(*
Nazwa:			GVL_Recipe
Opis:			Zmienne recepturowe tylko do wizualizacji
Wersja:			v0.2
Data:			2024-02-20
Autor:			MK
Urzadzenia:		
Konfiguracja:	
Info:
Zmiany:
- 20240220 [DP] Poprawki przed nowa wizką
*)
VAR_GLOBAL
	(*Legenda dla wizki :
		[H] - Hidden, prawdopodobnie nie potrzebne
		[I] - Info, informacja,
		[L] - Later, do zrobienia później, być może do przerobienia
		Uprawienia:
		brak opisu - operator
		[m] - Meechanik i powyżej
		[t] - Technolog i powyżej
		[s] - Serwis i powyżek
		[a] - Admin			
	*)	
	
	//Sorter nasadek, typ produktu	
	iCapSorterProductType										: INT		:= 2; 		//		Typ produktu: 0- kule/fliptopy, 1- pompki, 2- disctop, 3-airless, 4-decoration cap (wyłączone podcisnienie na załapywarce), 5- decoration cap with new gripper (wyłączone podcisnienie + nowy program do robota)
	uiCapSorterIndexShow										: UDINT		:= 5;		//		Index produktu	
	bPresenceBottleEnableShow									: BOOL;					//		Sprawdzanie butelki w formatce

//--------------------------------------CapSorterTransporter-----------------------------------------------------------------------------------------------------------------------------	
	// Sorter nasadek, transporter zasobnika
	bCapSorterTransporterEnableShow								: BOOL;					//		Aktywacja
	iCapSorterTransporterTankConveyorVelocityShow				: INT		:= 1200;	//		Prędkość 							| [%] (1.0-100.0)
	iCapSorterTransporterStartDelayTimeShow						: INT		:= 100;		//		Timer do załączania 				| [ms] (0.0-10_000.0)
	udiCapSorterTransporterTimeProductOnSensorBeforeBrushShow	: UDINT		:= 150;		//		Timer pracy							| [ms] (0.0-10_000.0)
	iCapSorterTransporterEmptyingConveyorSpeedShow				: INT		:= 25;		// 		Prędkość, opróżnianie 				| [%] (1.0-100.0)
	iCapSorterTransporterVolumeOfCapsShow						: INT		:= 330;		//		Odłegłość do zamknięć, ostrzeżenie 	| [mm] (0.0-10_000.0)

//---------------------------------------CapSorterWheel----------------------------------------------------------------------------------------------------------------------------	
	// Sorter nasadek, stól
	bCapSorterWheelEnableShow									: BOOL;					//		Aktywacja
	lrCapSorterWheelMoveAccelerationEmptyTableShow				: LREAL		:= 5000;	//		Dynamika rozpędzania - pusty 		| [obr/min²], (1.0-100_000.0) 
	lrCapSorterWheelMoveDecelerationEmptyTableShow				: LREAL		:= 5000;    //		Dynamika spowalniania - pusty 		| [obr/min²] (1.0-100_000.0) 
	lrCapSorterWheelMoveSpeedEmptyTableShow						: LREAL		:= 334;     //		Prędkość - pusty 					| [obr/min] (1.0-10_000.0)                
	lrCapSorterWheelMoveAngleEmptyTableShow						: LREAL		:= 20;      //		Kąt - pusty 						| [obr/min] (0.0-360.0)                        
	lrCapSorterWheelJerkAngleEmptyTableShow						: LREAL		:= 15000;   //		Zryw - pusty 						| [obr/min³] (1.0-1_000_000)                  
	iCapSorterWheelWaitingAfterRotationEmptyTableShow			: INT		:= 100;     //		Czas stabilizacji - pusty 			| [ms] (0.0-1_000)                 
	
	lrCapSorterWheelMoveAccelerationFullTableShow				: LREAL		:= 5000;	//		Dynamika rozpędzania - pełny 		| [obr/min²], (1.0-100_000.0) 
	lrCapSorterWheelMoveDecelerationFullTableShow				: LREAL		:= 5000;    //		Dynamika spowalniania - pełny 		| [obr/min²] (1.0-100_000.0) 
	lrCapSorterWheelMoveSpeedFullTableShow						: LREAL		:= 334;     //		Prędkość - pełny 					| [obr/min] (1.0-10_000.0)                
	lrCapSorterWheelMoveAngleFullyTableShow						: LREAL		:= 6;       //		Kąt - pełny 						| [obr/min] (0.0-360.0)                        
	lrCapSorterWheelJerkAngleFullTableShow						: LREAL		:= 15000;   //		Zryw - pełny 						| [obr/min³] (1.0-1_000_000)                  
	iCapSorterWheelWaitingAfterRotationFullTableShow			: INT		:= 30;      //		Czas stabilizacji - pełny 			| [ms] (0.0-1_000)                 
	
	lrCapSorterWheelMoveAccelerationHalfFullTableShow			: LREAL		:= 5000;	//		Dynamika rozpędzania - półpełny 	| [obr/min²], (1.0-100_000.0) 
	lrCapSorterWheelMoveDecelerationHalfFullTableShow			: LREAL		:= 5000;    //		Dynamika spowalniania - półpełny 	| [obr/min²] (1.0-100_000.0) 
	lrCapSorterWheelMoveSpeedHalfFullTableShow					: LREAL		:= 334;     //		Prędkość - półpełny 				| [obr/min] (1.0-10_000.0)                
	lrCapSorterWheelMoveAngleHalfFullyTableShow					: LREAL		:= 12;      //		Kąt - półpełny						| [obr/min] (0.0-360.0)                        
	lrCapSorterWheelJerkAngleHalfFullTableShow					: LREAL		:= 15000;   //		Zryw - półpełny 					| [obr/min³] (1.0-1_000_000)                  
	iCapSorterWheelWaitingAfterRotationHalfFullTableShow		: INT		:= 50;      //		Czas stabilizacji - półpełny 		| [ms] (0.0-1_000)               
	
//-------------------------------------CapSorterCamera------------------------------------------------------------------------------------------------------------------------------	                                                    	
	// Sorter nasadek, system wizyjny
	
    bCapSorterCameraEnableShow									: BOOL; 				//	[H]	Aktywacja                            	
	
//-----------------------------------------CapSorterRobot--------------------------------------------------------------------------------------------------------------------------	
	// Sorter nasadek, robot
	bCapSorterRobotEnableShow									: BOOL;					//		Aktywacja
                                                                                                                           	
	lrCapSorterRobotPlace1PositionXShow							: LREAL;				//		Offset odkładania 1, X 			| [mm]	((-100.0)-100.0)       
	lrCapSorterRobotPlace1PositionYShow							: lreal;    			//		Offset odkładania 1, Y 			| [mm]	((-100.0)-100.0)       
	lrCapSorterRobotPlace1PositionZShow							: lreal;    			//		Offset odkładania 1, Z 			| [mm]	((-100.0)-100.0)       
	lrCapSorterRobotPlace1PositionCShow							: lreal;    			//		Offset odkładania 1, C 			| [° ]	((-360.0)-360.0)                 
	iCapSorterRobotPickElevationShow							: INT;					//		Punkt nad poz. Pick				| [mm]	(30-1000)
	iCapSorterRobotPickTimeShow									: INT;					//		Czas przyssania					| [ms]	(0-10_000)
	iCapSorterRobotVacuumActivationShow							: INT;					//		Czas przed przyssaniem			| [ms]	(0-1000)
	iCapSorterRobotVacuumOffShow								: INT;					//		Czas przed oddmuchem			| [ms]	(0-1000)
	iCapSorterRobotPlaceTimeShow								: INT;					//		Czas oddmuchu					| [ms]	(0-1000)
	iCapSorterRobotTCP_PlaceOffsetShow							: INT;					//		Wysokość od TCP do p. odłożenia	| [mm]	(0-1000)									
	iCapSorterRobotAccelerationDecelerationShow					: INT;					//		Dynamika rozpędzania/hamowania	| [%]	(20-100)
	iCapSorterRobotGripperWatchdogShow							: INT;					//		Czas sprawdzania silownika		| [ms]	(0-1000)
	iCapSorterRobotParalaxCorrectionShow						: INT;					//		Korekta paralaxy				| [mm]	(0-100)
	
	iCapSorterRobotNumberToolShow								: INT;					//		Numer narzędzia					| 		(0-10)
	iCapSorterRobotPickPositionZShow							: INT;					//		Wysokość pobierania 			| [mm]	(0-200)
	iCapSorterRobotTCP_Lenght									: INT;					//		Długość chwytaka				| [mm]	(10-100)
	iCapSorterRobotProductDiametr								: INT;					//		Średnica nasadki				| [mm] 	(10-100)
	
//----------------------------------------CapSorterIntermediateTransporter---------------------------------------------------------------------------------------------------------------------------
	// Sorter nasadek, transporter zasypowy
	bCapSorterIntermediateTransporterEnableShow					: BOOL;					//		Aktywacja
	iCapSorterIntermediateTransporterAutoSpeedShow				: INT		:= 20;		//		Prędkość 					| [%] (1.0-100.0)
	iCapSorterIntermediateTransporterManualSpeedShow			: INT		:= 30;		//		Prędkość, manual 			| [%] (1.0-100.0)
	iCapSorterIntermediateTransporterEmptyingSpeedShow			: INT		:= 50;		//		Prędkość, opróżnianie 		| [%] (1.0-100.0)
	iCapSorterIntermediateTransporterDelayCountTimeShow			: INT		:= 100;		//		Timer pracy					| [ms]	(0.0-100_000.0)
	iCapSorterIntermediateTransporterReverseTimeShow			: INT		:= 4000;	//		Timer odwróconej pracy 		| [ms] (0.0-10_000.0)
	udiCapSorterIntermediateTransporterTimeProductOnSensorShow	: UDINT		:= 1800;	//		Czas produktu na czujniku 	| [ms] (0.0-10_000.0)	
	lrCapSorterIntermediateTransporterWheelAngleShow			: LREAL		:= 6;		//		Kąt zasypu 					| [°] (1.0-360.0)
	lrCapSorterIntermediateTransporterItemsSetValueShow			: LREAL	;				// 		Ilość detali na kołe		| []
	
//----------------------------------------CapSorterIntermediateBrush---------------------------------------------------------------------------------------------------------------------------
	//Sorter nasadek, szczotka transportera
	bCapSorterIntermediateBrushEnableShow						: BOOL;					//		Aktywacja
	iCapSorterIntermediateBrushAutoSpeedShow					: INT		:= 30;		//		Prędkość  					| [%] (0.0-100.0)
	iCapSorterIntermediateBrushManualSpeedShow					: INT		:= 30;		//		Prędkość, manual 			| [%] (0.0-100.0)
	iCapSorterIntermediateBrushEmptyingSpeedShow				: INT		:= 30;		//		Prędkość, opróżnianie 		| [%] (0.0-100.0)
	lrCapSorterIntermediateBrushPositionHeightSVShow			: LREAL		:= 45;		//		Wysokość 					| [mm] (0.0-10_000.0)

//----------------------------------------CapSorterBrush1OnWheel---------------------------------------------------------------------------------------------------------------------------
	// Sorter nasadek, szczotka stolu 1
	bCapSorterBrush1OnWheelEnableShow							: BOOL;					//		Aktywacja
	iCapSorterBrush1OnWheelAutoSpeedShow						: INT		:= 30;		//		Prędkość 					| [%] (0.0-100.0)
	iCapSorterBrush1OnWheelManualSpeedShow						: INT		:= 30;		//		Prędkość, manual 			| [%] (0.0-100.0)
	iCapSorterBrush1OnWheelEmptyingSpeedShow					: INT		:= 30;		//		Prędkość, opróżnianie 		| [%] (0.0-100.0)
	lrCapSorterBrush1OnWheelPositionHeightSVShow				: LREAL		:= 45;		//		Wysokość 					| [mm] (0.0-10_000.0)
	
//----------------------------------------CapSorterBrush2OnWheel----------------------------------------------------------------------------------
	// Sorter nasadek, szczotka stolu 2
	bCapSorterBrush2OnWheelEnableShow							: BOOL;					//		Aktywacja
	iCapSorterBrush2OnWheelAutoSpeedShow						: INT		:= 30;		//		Prędkość 					| [%] (0.0-100.0)
	iCapSorterBrush2OnWheelManualSpeedShow						: INT		:= 30;		//		Prędkość, manual 			| [%] (0.0-100.0)
	iCapSorterBrush2OnWheelEmptyingSpeedShow					: INT		:= 30;		//		Prędkość, opróżnianie 		| [%] (0.0-100.0)
	lrCapSorterBrush2OnWheelPositionHeightSVShow				: LREAL		:= 45;		//		Wysokość 					| [mm] (0.0-10_000.0)

//------------------------------------------CapFeeder-------------------------------------------------------------------------------------------------------------------------	
	// Sorter nasadek, 
	bCapSorterFeederEnableShow									: BOOL;					//		Aktywacjaa
	bCapSorterFeederEnableTubeError								: BOOL;					// 		Aktywacja błedu słomki
	lrCapSorterFeederMover1InputPositionShow					: LREAL;				//		Pozycja wkładania, wózek 1 	| [mm] (?-?)
	lrCapSorterFeederMover2InputPositionShow					: LREAL;				//		Pozycja wkładania, wózek 2 	| [mm] (?-?)
	lrCapSorterFeederMover1OutputPositionShow					: LREAL;				//		Pozycja wyjmowania, wózek 1 | [mm] (?-?)
	lrCapSorterFeederMover2OutputPositionShow					: LREAL;				//		Pozycja wyjmowania, wózek 2 | [mm] (?-?)
	lrCapSorterFeederSlotDistanceShow							: LREAL;				//		Offset wkładania			| [mm] (?-?)			Old-(Odstęp między pozycjami kładzenia)
	lrCapSorterFeederMoverSpeedShow								: LREAL;				//		Prędkość				 	| [%] (0.0-100.0)
	lrCapSorterFeederMoverAccelerationShow						: LREAL;				//		Przyspieszenie 				| [mm/s²] 
	lrCapSorterFeederMoveJerkShow								: LREAL;				//		Zryw						| [mm/s³]

//-------------------------------------------------------------------------------------------------------------------------------------------------------------------	
	//CapPreScrewer		
	bCapSorterPreScrewerEnableShow								: BOOL;					// 		Aktywacja
	bCapSorterPreScrewerPicker1EnableShow						: BOOL;					// 		Aktywacja	
	bCapSorterPreScrewerPicker2EnableShow						: BOOL;					// 		Aktywacja
	bCapSorterPreScrewerPicker3EnableShow						: BOOL;					// 		Aktywacja	
	bCapSorterPreScrewerPicker4EnableShow						: BOOL;					// 		Aktywacja
	//Oś Z
	lrCapSorterPreScrewerPickZPositionShow						: LREAL;				//		Wysokość pobierania						| [mm]	
	lrCapSorterPreScrewerCatcherReleseShow						: LREAL;				//		nie używamy Wysokość otwierania chwytaka nakrętek	| [mm]		
	lrCapSorterPreScrewerCapCatcherZPositionShow				: LREAL;				//		Wysokość zamykania nakrętkek			| [mm]
	lrCapSorterPreScrewerTopZPositionShow						: LREAL;				//		Pozycja górna ośi Z						| [mm] 	
	lrCapSorterPreScrewerCartesianCatchZPositionShow			: LREAL; 				//      Wait Position
	lrCapSorterPreScrewerStrawCatcherZPositionShow				: LREAL;				//		Wysokość otwierania łapaczy słomek		| [mm]	
	LrCapSorterPreScrewerCheckStrawCatcherActuatorZPosition		: LREAL;				//		Wysokość sparawdzania cofania łapaczy słomek	| [mm]	
	lrCapSorterPreScrewerScrewerStartZPositionShow				: LREAL;				//		Wysokość początku zakręcania			| [mm]	
	lrCapSorterPreScrewerGripperOpenPositionShow				: LREAL;				//		Pozycja otwierania chwytaka butelek 	| [mm]
	lrCapSorterPreScrewerPlaceZPositionShow						: LREAL;				//		Wysokość odkładania - koniec załapywania gwintu	| [mm] 

	lrCapSorterPreScrewerThreadPitchShow						: LREAL;				//		Skok gwintu 		| [mm]	
	lrCapSorterPreScrewerMultipleStartThreadShow				: LREAL;				//		Krotność gwintu
	lrCapSorterPreScrewerNumberOfThreadTurnsShow				: LREAL;				//		Ilość obrotów
  	
	//Wspólne ruchi	
	lrCapSorterPreScrewerBendingDistanceShow					: LREAL;				//		Odległość zaokrąglania ruchów 			| [mm]		
	lrCapSorterPreScrewerStrawInsertDistance					: LREAL;				//		Odległość wspólnego ruchu, prowadzenie słomki	| [mm]		
	//Oś x
	lrCapSorterPreScrewerPickXMover1PositionShow				: LREAL;				//		Pozycja osi poziomej do pobierania, wozek 1	| [mm]
	lrCapSorterPreScrewerPickXMover2PositionShow				: LREAL;				//		Pozycja osi poziomej do pobierania, wozek 2	| [mm]
	lrCapSorterPreScrewerPlaceXPositionShow						: LREAL;				//		Pozycja osi poziomej do odkładania			| [mm]
	//Oś zakręcania
	lrCapSorterPreScrewerScrewFindingShow						: LREAL;				//		Kąt szukania gwintu							| [°]
	lrCapSorterPreScrewerScrewDistanceShow						: LREAL;				//		Kąt zakręcania								| [°]
	//Prédkośći                                                                                                                         	
	lrCapSorterPreScrewerPickerSpeedShow						: LREAL;				//		Prędkość									| [%]   
	lrCapSorterPreScrewerPickerSpeedWhenScrewerShow				: LREAL;				//		Prędkość osi Z przy zakręcaniu				| [%]   
	lrCapSorterPreScrewerPickerAccelerationShow					: LREAL;				//		Przyspieszenie								| [mm/s²] 		
	lrCapSorterPreScrewerPickerJerkShow							: LREAL;				//		Zryw										| [mm/s³]
                                                                                                                                        	
	lrCapSorterPreScrewerCatcherSpeedShow						: LREAL;				//		Prędkość									| [mm/s] 
	lrCapSorterPreScrewerCatcherAccelerationShow				: LREAL;				//		Przyspieszenie								| [mm/s²] 	
	lrCapSorterPreScrewerCatcherJerkShow						: LREAL;				//		Zryw										| [mm/s³]	                                                                                                                                 	
	lrCapSorterPreScrewerScrewSpeedShow							: LREAL;				//		Prędkość zakręcania							| [mm/s]
	lrCapSorterPreScrewerScrewAccelerationShow					: LREAL;				//		Przyspieszenie zakręcania				| [mm/s²]
	lrCapSorterPreScrewerScrewJerkShow							: LREAL;				//		Zryw zakręcania							| [mm/s³]

	//Oś łapacza słomki	
	lrCapSorterPreScrewerCatcherCatchingPositionShow			: LREAL;				//		Pozycja łapania słomki					| [mm]
	lrCapSorterPreScrewerCatcherPlacePositionShow				: LREAL;				//		Pozycja dolna łapacza słomki			| [mm]
	lrCapSorterPreScrewerCatcherHightSVShow						: LREAL;				//		Nastawa wysokości stacji łapacza słomek		| [mm]
	//Kalibracja chwytaków butelki
	bCapSorterPreScrewerBottleCatcherEnableShow					: BOOL;					//		Actywacja chwytaków butelki
	lrCapSorterPreScrewerBottleCatch1OpenValueShow				: LREAL;				//		Chwytak 1 | wartość kalibracji otwartego chwytaka
	lrCapSorterPreScrewerBottleCatch1CloseValueShow				: LREAL;				//		Chwytak 1 | wartośc kalibracji zamkniętego chwytaka
	lrCapSorterPreScrewerBottleCatch2OpenValueShow				: LREAL;				//		Chwytak 2 | wartość kalibracji otwartego chwytaka
	lrCapSorterPreScrewerBottleCatch2CloseValueShow				: LREAL;				//		Chwytak 2 | wartość kalibracji zamkniętego chwytaka
	lrCapSorterPreScrewerBottleCatch3OpenValueShow				: LREAL;                //		Chwytak 3 | wartość kalibracji otwartego chwytaka
	lrCapSorterPreScrewerBottleCatch3CloseValueShow				: LREAL;				//		Chwytak 3 | wartość kalibracji zamkniętego chwytaka	
	lrCapSorterPreScrewerBottleCatch4OpenValueShow				: LREAL;                //		Chwytak 4 | wartość kalibracji otwartego chwytaka
	lrCapSorterPreScrewerBottleCatch4CloseValueShow				: LREAL;				//		Chwytak 4 | wartość kalibracji zamkniętego chwytaka
	                                                        	
	lrCapSorterPreScrewerBottleCatchToleranceValueShow			: LREAL;				//		Tolerancja chwytaków
	lrCapSorterPreScrewerCatchAngleOpenSV						: LREAL := 180.0;		//		[] Kąt puszczania centrowników
	
	lrCapSorterPreScrewerWaitInPlaceTimeShow					: LREAL	:= 50;			//		Czas zatrzymania w miejscu odłożenia 	| [ms]
	
	bCapSorterPreScrewerCatchAngleOpenEnaShow					: BOOL;					// 		Aktywacja puszczania centrowników po osiągnięciu zadanego kątu
	bCapSorterPreScrewerPoundedInCap							: BOOL;					// 		Wbijana nasadka
	
//Parametry do obliczeń 
	lrCapSorterBottleHightShow									: LREAL;				//		Wysokość butelki
	lrCapSorterBottleNeckHightShow								: LREAL;				// 		Wysokość szyjki butelki
	lrCapSorterCapHightShow										: LREAL;				// 		Wysokość zamknięcia
	lrCapSorterCapNeckHightShow									: LREAL;				//		Wysokość szyjki zamknięcia
	lrCapSorterPreScrewerCheckValveShow							: LREAL;				//		Długość zaworu zwrotnego				| [mm]
	
	lrCapSorterMoverHightShow									: LREAL := 226.0;		//		Wysokość wózków (Kartezjanem dotknąć ssawkami gniazdo do wkładania zamknięć)
	
//Rezerwa	
	lrCapSorterSpare1											: LREAL;				//Rezerwa 1
	lrCapSorterSpare2											: LREAL;				//Rezerwa 2
	lrCapSorterSpare3											: LREAL;				//Rezerwa 3
	lrCapSorterSpare4											: LREAL;				//Rezerwa 4
	lrCapSorterSpare5											: LREAL;				//Rezerwa 5
	lrCapSorterSpare6											: LREAL;				//Rezerwa 6
	lrCapSorterSpare7											: LREAL;				//Rezerwa 7	
	
	
	
END_VAR

(* stored: Version 1.2.0.0, ProductVersion 3.1.4026.13, FileIdentifier 6263720f6917e4e146896e1f81689e527645a13a, FileSignature 9c40f417a2ccb9bccc81df56e038249afd327ee3ea36e480ff7fc71d07a767fa5d43ace40f54f1f42967ae730aa4b43b460ffa6d5cef69fca09d12e5450bfe0f227af3b9e8a04afce32d2bd4ac08b3e040de7c29d727209f2b3505aff9e45a12874c65b4abcfb1b8f42560ac0d48a7d5ff1fc99ce8d712edc4426d085ea97ae6ee183b23daf1bda230cce1964f0a3d01c69072917108922f167891ca29bd3b4f64cb5fdb313a96852c5450ac7848886452df9b1aa11ffcc1a14a35e2bb79385d5facb35bc5fa7ba611a4d0e2ff282382f5ee38976cf9b0e69aa0076699aa63f5127385e9cc6a0ea836e6f015d5e9dd0d9314c4f07ebe086addccbc73928ad300
   GVL GVL_Recipe: Id {7a794286-5358-476a-aa62-1dd70bbc5105} *)
